# B&R Automation Studio project MiRepo
Automation Studio 4.7.6.114 SP; technology packages: mapp 5.6.2

## Configuration Config1

CPU 4PPC70.101G-20B, AutomationRuntime C4.72, Build 4.1.2, Vc V4.72.0

### Task classes (Cpu.sw)
```
Cyclic#4:
  Main <- Source.Main.prg
  ControlPue <- Source.ControlPuertas.prg
VcDataObjects: Visu <- Visu.Visu.dob
Libraries: standard
```

### Hardware
```
4PPC70_101G_20B : 4PPC70.101G-20B v1.5.0.1
  Connector IF2:
    ActivateDevice = 1
  VcObjectName = Visu
  KeyMappingFile = VC\4PPC70_101G_20B.dis
```

### Config.mpalarmxcore - 4PPC70_101G_20B/mappServices/Config.mpalarmxcore
```
Element gMpAlarmXCore (Type=mpalarmxcore)
  mapp.AlarmX.Core.Configuration:
    [0]:
      Name = Alarma 1
      Message = Esta es una alarma de ejemplo
```

## Logical view

Binary libraries used (declarations not repeated): operator, runtime, astime, AsIecCon, standard, MpAlarmX 5.06.2, MpBase 5.06.0

### Global.typ - Global data types
```iecst
TYPE
	Main_ctrl_type : 	STRUCT
		cmd : USINT;
		param : USINT;
		status : USINT;
		state : USINT;
	END_STRUCT;
END_TYPE
```

### Global.var - Global variables
```iecst
VAR
	gCtrl : Main_ctrl_type;
END_VAR
```


### Program Logical/Source/Main (IEC)

#### Types.typ
```iecst
TYPE
	New_Enumeration2 :
		(
		New_Member
		);
	New_Enumeration1 :
		(
		New_Member1
		);
	New_Enumeration :
		(
		New_Member2
		);
END_TYPE
```

#### Variables.var
```iecst
VAR
	ok : BOOL;
	puerta : BOOL;
	state : INT;
END_VAR
```

#### Main.st
```iecst
PROGRAM _INIT
	//Inicialización
	ok := FALSE;
	puerta := FALSE;

END_PROGRAM

PROGRAM _CYCLIC

	IF ok THEN
		puerta := TRUE;
	END_IF;

	// Hola mundo del GIT

END_PROGRAM
```

### Program Logical/Source/ControlPuertas (IEC)

#### Cyclic.ld - Cyclic code
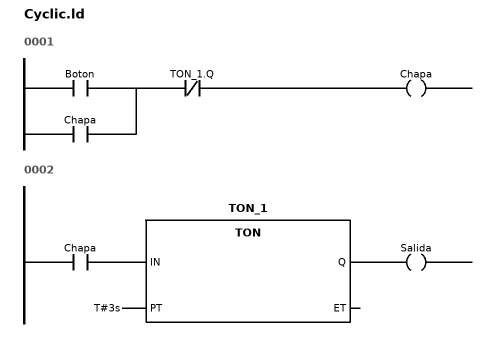
Ladder, written as Structured Text:
```iecst
PROGRAM _CYCLIC
(* Network 1 *)
Chapa := (Boton OR Chapa) AND NOT TON_1.Q;

(* Network 2 *)
TON_1(IN := Chapa, PT := T#3s);
Salida := TON_1.Q;
END_PROGRAM
```

#### Variables.var - Local variables
```iecst
VAR
	Boton : BOOL;
	Chapa : BOOL;
	TON_1 : TON;
	Salida : BOOL;
END_VAR
```

- Visualisation Logical/Visu (not shown)

Listed in the project but not available here: Logical/Source/ControlPuertas/Init.ld, Logical/Source/ControlPuertas/Types.typ
